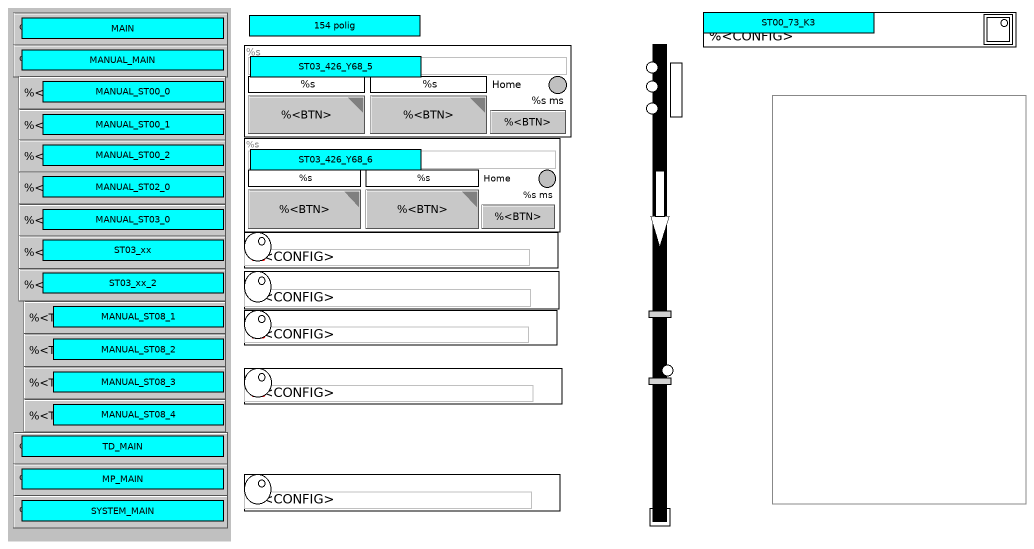
[picture p118: MANUAL_ST03_4 (HMI screen)]
embedded screen at (3,115)-(226,648): M0000_Manual
embedded screen at (239,152)-(566,244): ZLIB_VALVE_1_SENSORS
embedded screen at (239,245)-(555,339): ZLIB_VALVE_1_SENSORS
embedded screen at (239,417)-(552,452): VDIGIN
embedded screen at (239,339)-(553,375): VDIGIN
embedded screen at (239,378)-(554,416): VDIGIN
embedded screen at (239,581)-(555,618): VDIGIN
embedded screen at (239,475)-(557,511): VDIGIN
embedded screen at (636,151)-(677,633): ZUFUEHRUNG_154POL; invisible if gTypeCode<>4871
rectangle at (244,122)-(415,143): text "154 polig"; invisible if TRUE
rectangle at (245,163)-(416,184): text "ST03_426_Y68_5"; invisible if TRUE
rectangle at (245,256)-(416,277): text "ST03_426_Y68_6"; invisible if TRUE
embedded screen at (698,119)-(1011,154): VDIGOUT_SMAL
rectangle at (698,119)-(869,140): text "ST00_73_K3"; invisible if TRUE
1 more shapes without text or variables
*)

(* Visualisation MANUAL_ST03_5
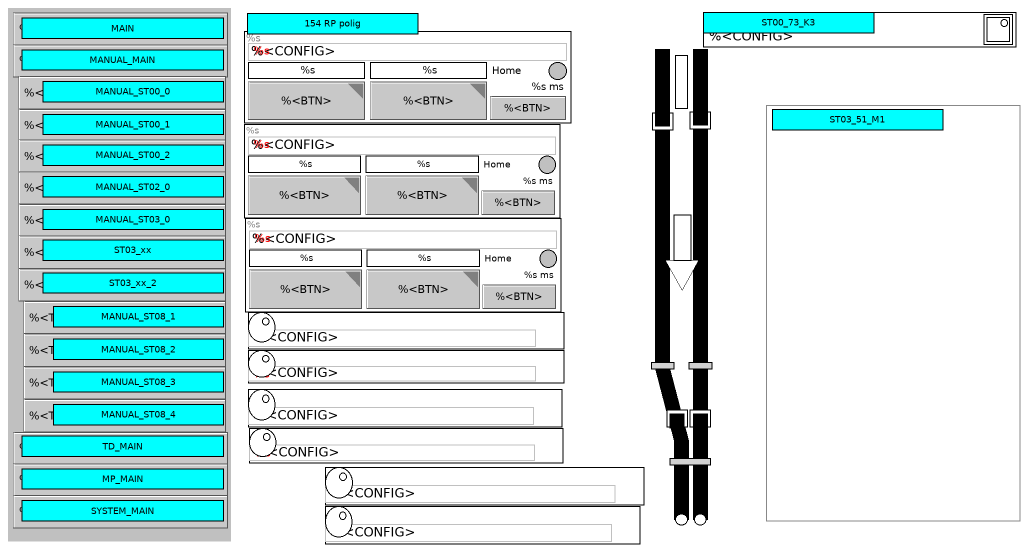
embedded screen at (3,115)-(226,648): M0000_Manual
embedded screen at (239,138)-(566,230): ZLIB_VALVE_1_SENSORS
embedded screen at (239,231)-(555,325): ZLIB_VALVE_1_SENSORS
embedded screen at (244,535)-(558,570): VDIGIN
embedded screen at (320,574)-(639,612): VDIGIN
embedded screen at (243,457)-(559,490): VDIGIN
embedded screen at (243,496)-(557,534): VDIGIN
embedded screen at (243,419)-(559,456): VDIGIN
embedded screen at (320,613)-(635,651): VDIGIN
embedded screen at (240,325)-(556,419): ZLIB_VALVE_1_SENSORS
embedded screen at (646,156)-(707,632): ZUFUEHRUNG_154RP; invisible if gTypeCode<>4872
rectangle at (242,120)-(413,141): text "154 RP polig"; invisible if TRUE
rectangle at (767,216)-(938,237): text "ST03_51_M1"; invisible if TRUE
embedded screen at (698,119)-(1011,154): VDIGOUT_SMAL
rectangle at (698,119)-(869,140): text "ST00_73_K3"; invisible if TRUE
1 more shapes without text or variables
*)

(* Visualisation MANUAL_ST03_6
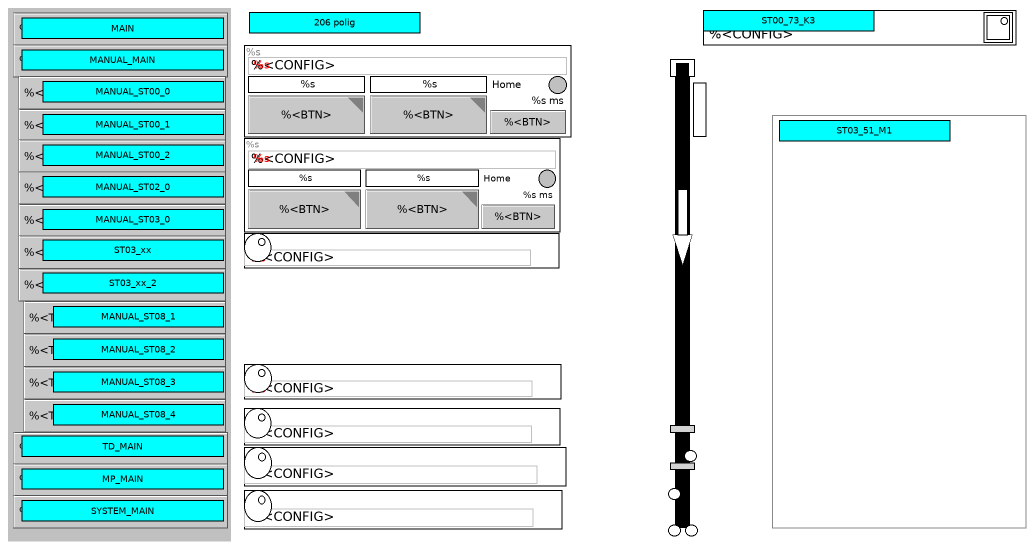
embedded screen at (3,115)-(226,648): M0000_Manual
embedded screen at (239,152)-(566,244): ZLIB_VALVE_1_SENSORS
embedded screen at (239,245)-(555,339): ZLIB_VALVE_1_SENSORS
embedded screen at (239,554)-(561,593): VDIGIN
embedded screen at (239,340)-(554,375): VDIGIN
embedded screen at (239,515)-(555,552): VDIGIN
embedded screen at (239,597)-(557,636): VDIGIN
embedded screen at (239,471)-(556,506): VDIGIN
embedded screen at (646,161)-(701,643): ZUFUEHRUNG_206POL; invisible if gTypeCode<>522
rectangle at (244,119)-(415,140): text "206 polig"; invisible if TRUE
rectangle at (774,227)-(945,248): text "ST03_51_M1"; invisible if TRUE
embedded screen at (698,117)-(1011,152): VDIGOUT_SMAL
rectangle at (698,117)-(869,138): text "ST00_73_K3"; invisible if TRUE
1 more shapes without text or variables
*)

(* Visualisation MANUAL_ST03_7
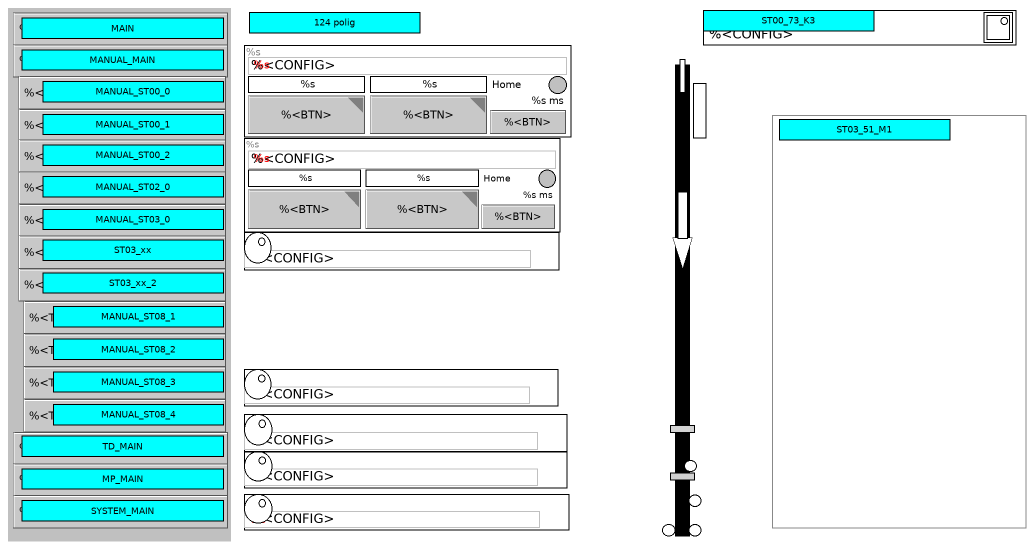
embedded screen at (3,115)-(226,648): M0000_Manual
embedded screen at (239,152)-(566,244): ZLIB_VALVE_1_SENSORS
embedded screen at (239,245)-(555,339): ZLIB_VALVE_1_SENSORS
embedded screen at (239,558)-(562,595): VDIGIN
embedded screen at (239,339)-(554,377): VDIGIN
embedded screen at (239,521)-(562,559): VDIGIN
embedded screen at (239,601)-(564,637): VDIGIN
embedded screen at (239,476)-(553,513): VDIGIN
embedded screen at (646,161)-(701,643): ZUFUEHRUNG_124POL; invisible if gTypeCode<>564
rectangle at (244,119)-(415,140): text "124 polig"; invisible if TRUE
rectangle at (774,226)-(945,247): text "ST03_51_M1"; invisible if TRUE
embedded screen at (698,117)-(1011,152): VDIGOUT_SMAL
rectangle at (698,117)-(869,138): text "ST00_73_K3"; invisible if TRUE
1 more shapes without text or variables
*)

(* Visualisation MANUAL_ST03_8
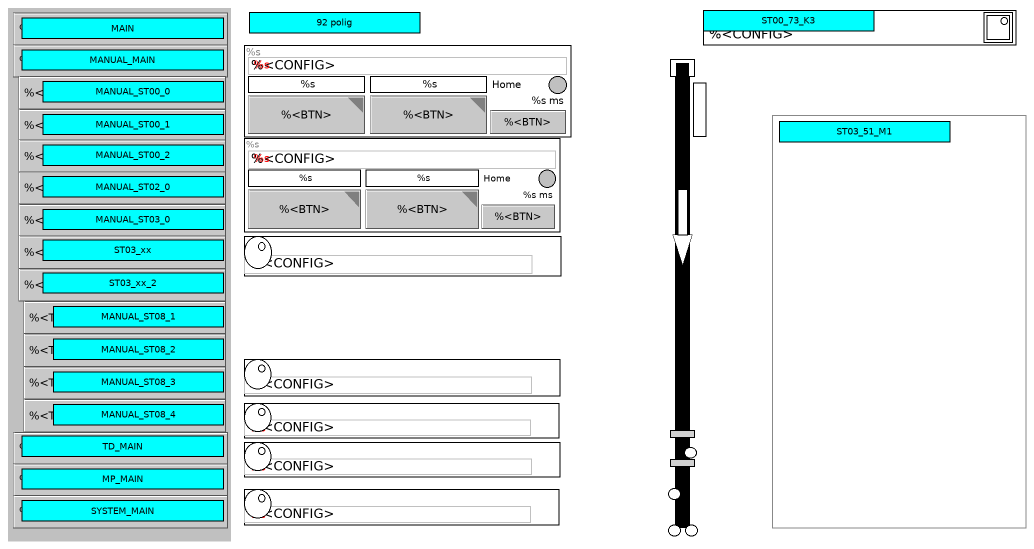
embedded screen at (3,115)-(226,648): M0000_Manual
embedded screen at (239,152)-(566,244): ZLIB_VALVE_1_SENSORS
embedded screen at (239,245)-(555,339): ZLIB_VALVE_1_SENSORS
embedded screen at (239,549)-(555,584): VDIGIN
embedded screen at (239,343)-(556,383): VDIGIN
embedded screen at (239,510)-(554,545): VDIGIN
embedded screen at (239,596)-(554,632): VDIGIN
embedded screen at (239,466)-(555,503): VDIGIN
embedded screen at (646,161)-(701,643): ZUFUEHRUNG_92POL; invisible if gTypeCode<>550
rectangle at (244,119)-(415,140): text "92 polig"; invisible if TRUE
rectangle at (774,228)-(945,249): text "ST03_51_M1"; invisible if TRUE
embedded screen at (698,117)-(1011,152): VDIGOUT_SMAL
rectangle at (698,117)-(869,138): text "ST00_73_K3"; invisible if TRUE
1 more shapes without text or variables
*)

(* Visualisation MANUAL_ST03_9
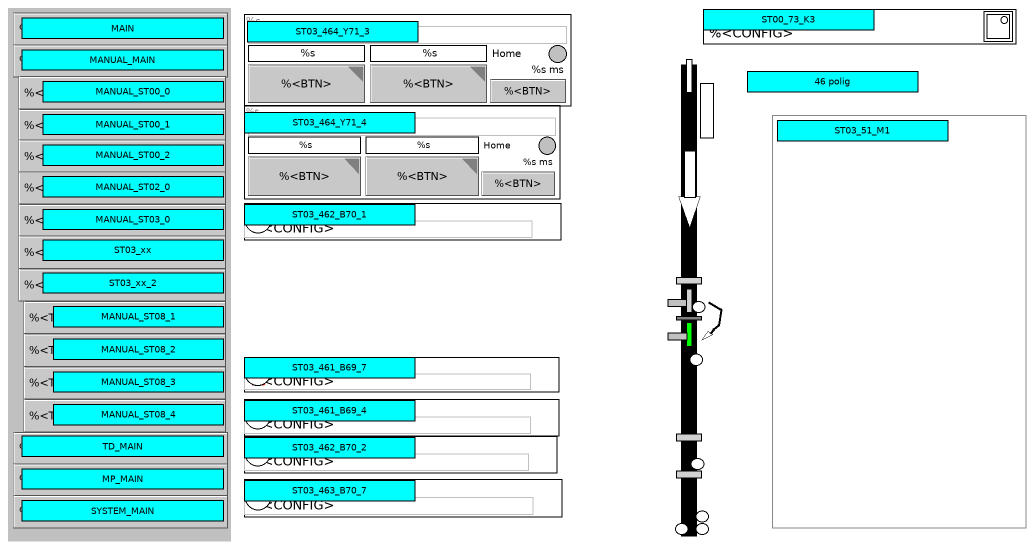
embedded screen at (3,115)-(226,648): M0000_Manual
embedded screen at (239,121)-(566,213): ZLIB_VALVE_1_SENSORS
embedded screen at (239,212)-(555,306): ZLIB_VALVE_1_SENSORS
embedded screen at (239,543)-(552,580): VDIGIN
embedded screen at (239,310)-(556,347): VDIGIN
embedded screen at (239,506)-(554,543): VDIGIN
embedded screen at (239,586)-(557,624): VDIGIN
embedded screen at (239,464)-(554,499): VDIGIN
embedded screen at (646,161)-(716,643): ZUFUEHRUNG_46POL; invisible if gTypeCode<>569
rectangle at (742,178)-(913,199): text "46 polig"; invisible if TRUE
rectangle at (239,219)-(410,240): text "ST03_464_Y71_4"; invisible if TRUE
rectangle at (242,128)-(413,149): text "ST03_464_Y71_3"; invisible if TRUE
rectangle at (239,311)-(410,332): text "ST03_462_B70_1"; invisible if TRUE
rectangle at (239,507)-(410,528): text "ST03_461_B69_4"; invisible if TRUE
rectangle at (239,544)-(410,565): text "ST03_462_B70_2"; invisible if TRUE
rectangle at (239,587)-(410,608): text "ST03_463_B70_7"; invisible if TRUE
rectangle at (239,464)-(410,485): text "ST03_461_B69_7"; invisible if TRUE
rectangle at (772,227)-(943,248): text "ST03_51_M1"; invisible if TRUE
embedded screen at (698,116)-(1011,151): VDIGOUT_SMAL
rectangle at (698,116)-(869,137): text "ST00_73_K3"; invisible if TRUE
1 more shapes without text or variables
*)

(* Visualisation MANUAL_ST03_9_2
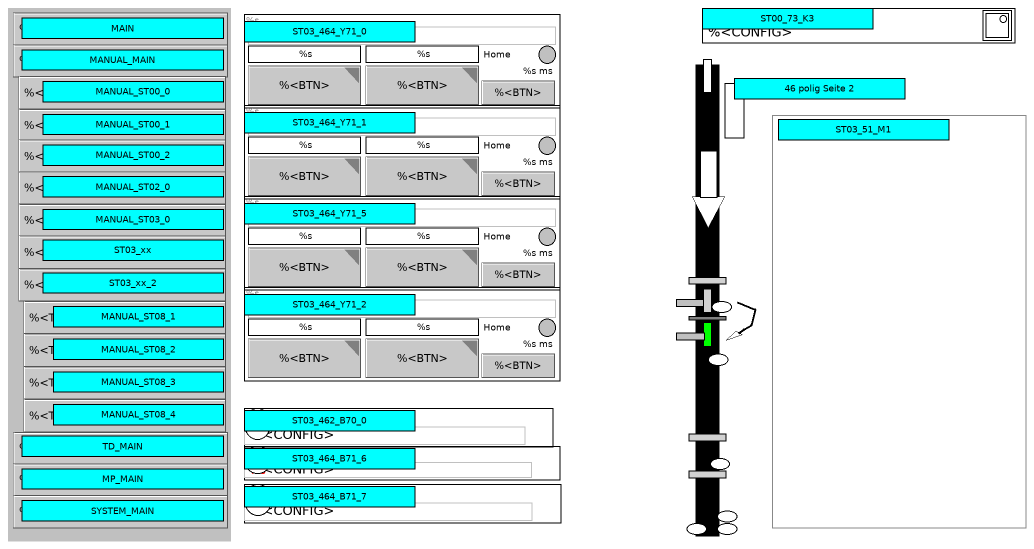
embedded screen at (3,115)-(226,648): M0000_Manual
embedded screen at (646,161)-(750,643): ZUFUEHRUNG_46POL; invisible if gTypeCode<>569
rectangle at (729,185)-(900,206): text "46 polig Seite 2"; invisible if TRUE
embedded screen at (239,553)-(555,587): VDIGIN
embedded screen at (239,121)-(555,215): ZLIB_VALVE_1_SENSORS
rectangle at (239,128)-(410,149): text "ST03_464_Y71_0"; invisible if TRUE
rectangle at (239,555)-(410,576): text "ST03_464_B71_6"; invisible if TRUE
embedded screen at (239,212)-(555,306): ZLIB_VALVE_1_SENSORS
rectangle at (239,219)-(410,240): text "ST03_464_Y71_1"; invisible if TRUE
embedded screen at (239,394)-(555,488): ZLIB_VALVE_1_SENSORS
rectangle at (239,401)-(410,422): text "ST03_464_Y71_2"; invisible if TRUE
embedded screen at (239,303)-(555,397): ZLIB_VALVE_1_SENSORS
rectangle at (239,310)-(410,331): text "ST03_464_Y71_5"; invisible if TRUE
embedded screen at (239,515)-(548,554): VDIGIN
rectangle at (239,517)-(410,538): text "ST03_462_B70_0"; invisible if TRUE
rectangle at (773,226)-(944,247): text "ST03_51_M1"; invisible if TRUE
embedded screen at (239,591)-(556,630): VDIGIN
rectangle at (239,593)-(410,614): text "ST03_464_B71_7"; invisible if TRUE
embedded screen at (697,115)-(1010,150): VDIGOUT_SMAL
rectangle at (697,115)-(868,136): text "ST00_73_K3"; invisible if TRUE
1 more shapes without text or variables
*)

(* Visualisation MANUAL_ST08_1
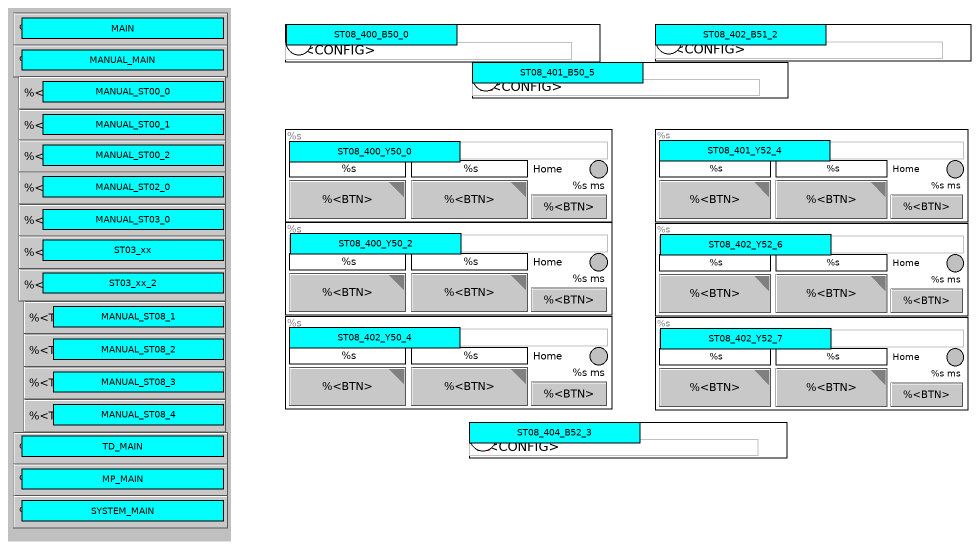
embedded screen at (3,115)-(226,648): M0000_Manual
embedded screen at (280,236)-(607,329): ZLIB_VALVE_1_SENSORS; invisible if NOT .MP.ST08.Trayzufuhr_Verlaengerung
embedded screen at (280,329)-(607,422): ZLIB_VALVE_1_SENSORS
embedded screen at (280,131)-(595,169): VDIGIN
embedded screen at (467,169)-(783,205): VDIGIN
embedded screen at (650,131)-(966,168): VDIGIN
embedded screen at (280,423)-(607,516): ZLIB_VALVE_1_SENSORS
embedded screen at (650,236)-(963,329): ZLIB_VALVE_1_SENSORS; invisible if NOT .MP.ST08.Traystapel_schieben OR NOT .MP.ST08.Trayzufuhr_Verlaengerung
embedded screen at (650,330)-(963,423): ZLIB_VALVE_1_SENSORS; invisible if NOT .MP.ST08.Traystapel_schieben OR NOT .MP.ST08.Trayzufuhr_Verlaengerung
embedded screen at (650,424)-(963,517): ZLIB_VALVE_1_SENSORS; invisible if NOT .MP.ST08.Traystapel_schieben
embedded screen at (464,529)-(782,565): VDIGIN
rectangle at (281,131)-(452,152): text "ST08_400_B50_0"; invisible if TRUE
rectangle at (467,169)-(638,190): text "ST08_401_B50_5"; invisible if TRUE
rectangle at (650,131)-(821,152): text "ST08_402_B51_2"; invisible if TRUE
rectangle at (284,248)-(455,269): text "ST08_400_Y50_0"; invisible if TRUE
rectangle at (285,340)-(456,361): text "ST08_400_Y50_2"; invisible if TRUE
rectangle at (654,247)-(825,268): text "ST08_401_Y52_4"; invisible if TRUE
rectangle at (655,341)-(826,362): text "ST08_402_Y52_6"; invisible if TRUE
rectangle at (655,435)-(826,456): text "ST08_402_Y52_7"; invisible if TRUE
rectangle at (284,434)-(455,455): text "ST08_402_Y50_4"; invisible if TRUE
rectangle at (464,529)-(635,550): text "ST08_404_B52_3"; invisible if TRUE
*)

(* Visualisation MANUAL_ST08_2
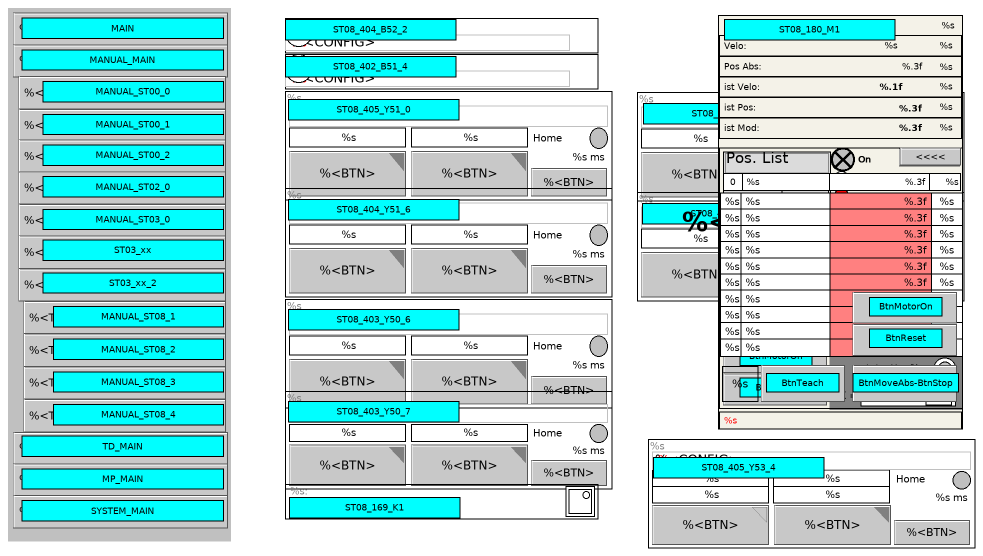
embedded screen at (3,115)-(226,648): M0000_Manual
embedded screen at (280,125)-(593,160): VDIGIN
embedded screen at (280,198)-(607,307): ZLIB_VALVE_1_SENSORS
embedded screen at (280,295)-(607,404): ZLIB_VALVE_1_SENSORS
embedded screen at (643,546)-(970,655): ZLIB_VALVE_2_SENSORS
embedded screen at (280,406)-(607,515): ZLIB_VALVE_1_SENSORS
embedded screen at (280,498)-(607,596): ZLIB_VALVE_1_SENSORS
embedded screen at (280,161)-(593,196): VDIGIN
embedded screen at (632,199)-(959,308): ZLIB_VALVE_1_SENSORS; invisible if MP.ST08.StapelMotor
rectangle at (638,210)-(809,231): text "ST08_404_Y53_0"; invisible if TRUE
embedded screen at (632,299)-(959,408): ZLIB_VALVE_1_SENSORS; invisible if MP.ST08.StapelMotor
rectangle at (637,310)-(808,331): text "ST08_404_Y53_2"; invisible if TRUE
embedded screen at (713,122)-(959,536): ZLIB_7211_Achse; invisible if NOT MP.ST08.StapelMotor
embedded screen at (280,591)-(593,626): VDIGOUT_SMAL
rectangle at (280,126)-(451,147): text "ST08_404_B52_2"; invisible if TRUE
rectangle at (280,163)-(451,184): text "ST08_402_B51_4"; invisible if TRUE
rectangle at (283,206)-(454,227): text "ST08_405_Y51_0"; invisible if TRUE
rectangle at (283,306)-(454,327): text "ST08_404_Y51_6"; invisible if TRUE
rectangle at (283,416)-(454,437): text "ST08_403_Y50_6"; invisible if TRUE
rectangle at (283,508)-(454,529): text "ST08_403_Y50_7"; invisible if TRUE
rectangle at (284,604)-(455,625): text "ST08_169_K1"; invisible if TRUE
rectangle at (648,564)-(819,585): text "ST08_405_Y53_4"; invisible if TRUE
rectangle at (719,126)-(890,147): text "ST08_180_M1"; invisible if TRUE
*)

(* Visualisation MANUAL_ST08_3
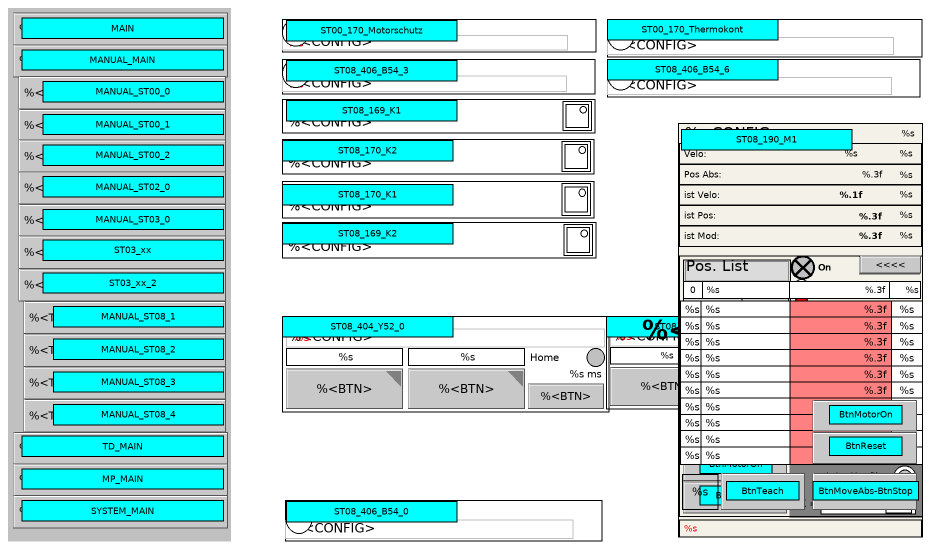
embedded screen at (3,115)-(226,648): M0000_Manual
embedded screen at (277,206)-(590,240): VDIGOUT_SMAL
embedded screen at (277,329)-(591,365): VDIGOUT_SMAL
embedded screen at (277,288)-(589,325): VDIGOUT_SMAL
embedded screen at (277,246)-(589,281): VDIGOUT_SMAL
embedded screen at (602,126)-(917,164): VDIGIN
embedded screen at (277,126)-(591,159): VDIGIN
embedded screen at (280,607)-(597,648): VDIGIN
embedded screen at (277,166)-(590,201): VDIGIN
embedded screen at (601,423)-(914,516): ZLIB_VALVE_1_SENSORS; invisible if MP.ST08.TrayAushebenMotor
embedded screen at (277,423)-(604,519): ZLIB_VALVE_1_SENSORS
rectangle at (601,423)-(772,444): text "ST08_406_Y52_3"; invisible if TRUE
rectangle at (277,423)-(448,444): text "ST08_404_Y52_0"; invisible if TRUE
rectangle at (281,207)-(452,228): text "ST08_169_K1"; invisible if TRUE
rectangle at (277,330)-(448,351): text "ST08_169_K2"; invisible if TRUE
rectangle at (277,291)-(448,312): text "ST08_170_K1"; invisible if TRUE
rectangle at (277,247)-(448,268): text "ST08_170_K2"; invisible if TRUE
rectangle at (281,127)-(452,148): text "ST00_170_Motorschutz"; invisible if TRUE
rectangle at (602,126)-(773,147): text "ST00_170_Thermokont"; invisible if TRUE
rectangle at (281,608)-(452,629): text "ST08_406_B54_0"; invisible if TRUE
rectangle at (281,167)-(452,188): text "ST08_406_B54_3"; invisible if TRUE
embedded screen at (602,166)-(915,204): VDIGIN
rectangle at (602,166)-(773,187): text "ST08_406_B54_6"; invisible if TRUE
embedded screen at (673,230)-(919,644): ZLIB_7211_Achse; invisible if NOT MP.ST08.TrayAushebenMotor
rectangle at (676,236)-(847,257): text "ST08_190_M1"; invisible if TRUE
*)

(* Visualisation MANUAL_ST08_4
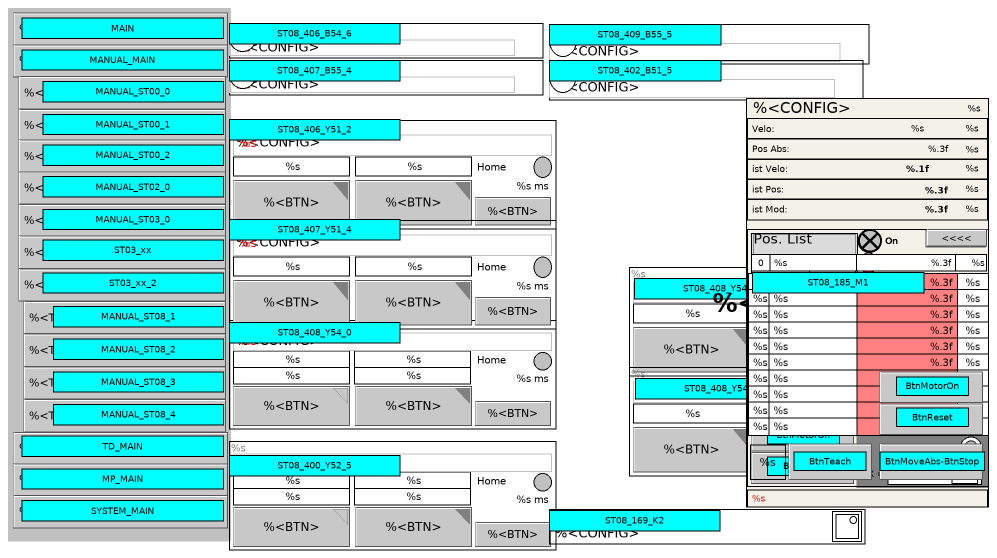
embedded screen at (3,115)-(226,648): M0000_Manual
embedded screen at (224,427)-(551,536): ZLIB_VALVE_2_SENSORS
embedded screen at (224,130)-(538,165): VDIGIN
embedded screen at (224,227)-(551,336): ZLIB_VALVE_1_SENSORS
embedded screen at (224,327)-(551,436): ZLIB_VALVE_1_SENSORS
embedded screen at (544,131)-(864,171): VDIGIN
embedded screen at (224,548)-(551,657): ZLIB_VALVE_2_SENSORS; invisible if MP.ST03.SGM_3621
embedded screen at (544,167)-(858,207): VDIGIN
embedded screen at (624,374)-(951,483): ZLIB_VALVE_1_SENSORS; invisible if MP.ST08.StapelMotor
rectangle at (629,385)-(801,406): text "ST08_408_Y54_2"; invisible if TRUE
embedded screen at (624,474)-(951,583): ZLIB_VALVE_1_SENSORS; invisible if MP.ST08.StapelMotor
rectangle at (630,485)-(802,506): text "ST08_408_Y54_4"; invisible if TRUE
embedded screen at (741,205)-(985,614): ZLIB_7211_Achse; invisible if NOT MP.ST08.StapelMotor
embedded screen at (224,167)-(538,202): VDIGIN
embedded screen at (544,616)-(860,651): VDIGOUT_SMAL
rectangle at (224,562)-(395,583): text "ST08_400_Y52_5"; invisible if TRUE
rectangle at (544,617)-(715,638): text "ST08_169_K2"; invisible if TRUE
rectangle at (224,429)-(395,450): text "ST08_408_Y54_0"; invisible if TRUE
rectangle at (224,326)-(395,347): text "ST08_407_Y51_4"; invisible if TRUE
rectangle at (224,226)-(395,247): text "ST08_406_Y51_2"; invisible if TRUE
rectangle at (224,130)-(395,151): text "ST08_406_B54_6"; invisible if TRUE
rectangle at (224,167)-(395,188): text "ST08_407_B55_4"; invisible if TRUE
rectangle at (544,131)-(716,152): text "ST08_409_B55_5"; invisible if TRUE
rectangle at (544,167)-(716,188): text "ST08_402_B51_5"; invisible if TRUE
rectangle at (747,379)-(919,400): text "ST08_185_M1"; invisible if TRUE
*)

(* Visualisation DIALOG_SAVE_AS
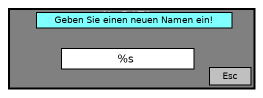
rectangle at (1,0)-(248,81): text "%<DATA>"; shows 'save_as'
rectangle at (54,40)-(187,61): text "%s"; shows $InputVar$; invisible if ( *NOT ST_TD.b_Dialog_save_as_on* ); editable
rectangle at (29,4)-(225,20): text "Geben Sie einen neuen Namen ein!"; invisible if TRUE
rectangle at (202,59)-(244,77): text "Esc"; toggles TDHandler.b_Dialog_save_as_on
*)

(* Visualisation TD_01_EDIT
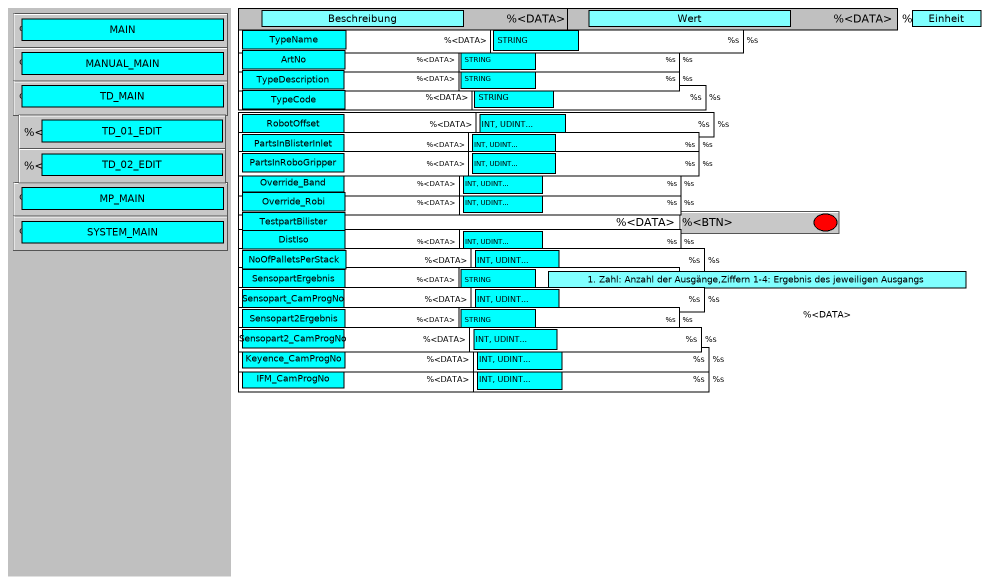
embedded screen at (3,115)-(226,683): M0003_TD
rectangle at (796,407)-(1009,436): text "%<DATA>"; shows 'Info_01'; invisible if gTypeCode<>4991 AND gTypeCode <>312
embedded screen at (233,317)-(834,342): Data_BOOL
embedded screen at (233,192)-(870,217): Data_STRING
embedded screen at (233,297)-(834,322): Data_DEZIMAL
embedded screen at (233,278)-(834,303): Data_DEZIMAL
embedded screen at (233,173)-(834,198): Data_STRING
embedded screen at (233,154)-(834,179): Data_STRING
embedded screen at (233,135)-(921,160): Data_STRING
embedded screen at (233,336)-(834,361): Data_DEZIMAL
embedded screen at (233,355)-(866,380): Data_DEZIMAL
embedded screen at (233,374)-(834,399): Data_STRING
rectangle at (237,137)-(341,156): text "TypeName"; invisible if TRUE
rectangle at (237,157)-(340,176): text "ArtNo"; invisible if TRUE
rectangle at (237,177)-(339,196): text "TypeDescription"; invisible if TRUE
rectangle at (237,197)-(340,216): text "TypeCode"; invisible if TRUE
rectangle at (237,280)-(339,299): text "Override_Band"; invisible if TRUE
rectangle at (237,299)-(340,318): text "Override_Robi"; invisible if TRUE
rectangle at (237,319)-(340,338): text "TestpartBilister"; invisible if TRUE
rectangle at (237,337)-(340,356): text "DistIso"; invisible if TRUE
rectangle at (237,376)-(340,395): text "SensopartErgebnis"; invisible if TRUE
rectangle at (237,357)-(341,376): text "NoOfPalletsPerStack"; invisible if TRUE
rectangle at (543,378)-(961,395): text "1. Zahl: Anzahl der Ausgänge,Ziffern 1-4: Ergebnis des jeweiligen Ausgangs"; invisible if TRUE
embedded screen at (233,219)-(879,244): Data_DEZIMAL
rectangle at (237,221)-(339,240): text "RobotOffset"; invisible if TRUE
embedded screen at (233,239)-(859,264): Data_DEZIMAL
rectangle at (237,241)-(339,260): text "PartsInBlisterInlet"; invisible if TRUE
embedded screen at (233,474)-(872,499): Data_DEZIMAL
rectangle at (237,476)-(339,495): text "IFM_CamProgNo"; invisible if TRUE
embedded screen at (233,394)-(866,419): Data_DEZIMAL
rectangle at (237,396)-(339,415): text "Sensopart_CamProgNo"; invisible if TRUE
embedded screen at (233,258)-(859,283): Data_DEZIMAL
rectangle at (237,260)-(339,279): text "PartsInRoboGripper"; invisible if TRUE
embedded screen at (233,115)-(987,137): DATA_HEADER_BEER
embedded screen at (233,454)-(872,479): Data_DEZIMAL
rectangle at (237,456)-(340,475): text "Keyence_CamProgNo"; invisible if TRUE
embedded screen at (233,414)-(834,439): Data_STRING
rectangle at (237,416)-(340,435): text "Sensopart2Ergebnis"; invisible if TRUE
embedded screen at (233,434)-(862,459): Data_DEZIMAL
rectangle at (237,436)-(339,455): text "Sensopart2_CamProgNo"; invisible if TRUE
*)

(* Visualisation TD_02_EDIT
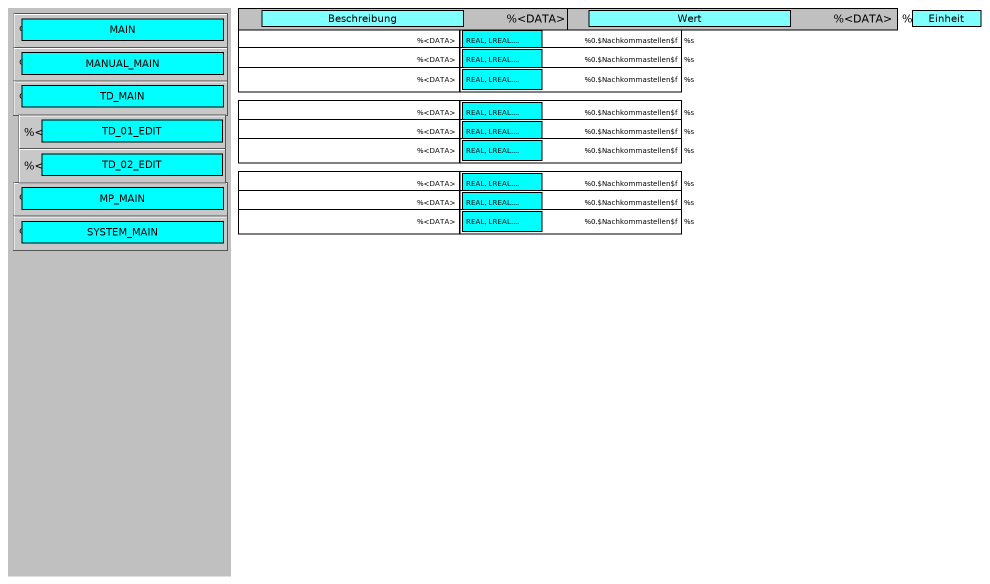
embedded screen at (3,115)-(226,683): M0003_TD
embedded screen at (233,135)-(834,160): Data_DEZIMAL_REAL
embedded screen at (233,154)-(834,179): Data_DEZIMAL_REAL
embedded screen at (233,174)-(834,199): Data_DEZIMAL_REAL
embedded screen at (233,207)-(834,232): Data_DEZIMAL_REAL
embedded screen at (233,226)-(834,251): Data_DEZIMAL_REAL
embedded screen at (233,245)-(834,270): Data_DEZIMAL_REAL
embedded screen at (233,115)-(987,137): DATA_HEADER_BEER
embedded screen at (233,278)-(834,303): Data_DEZIMAL_REAL
embedded screen at (233,297)-(834,322): Data_DEZIMAL_REAL
embedded screen at (233,316)-(834,341): Data_DEZIMAL_REAL
*)

(* Visualisation TD_MAIN
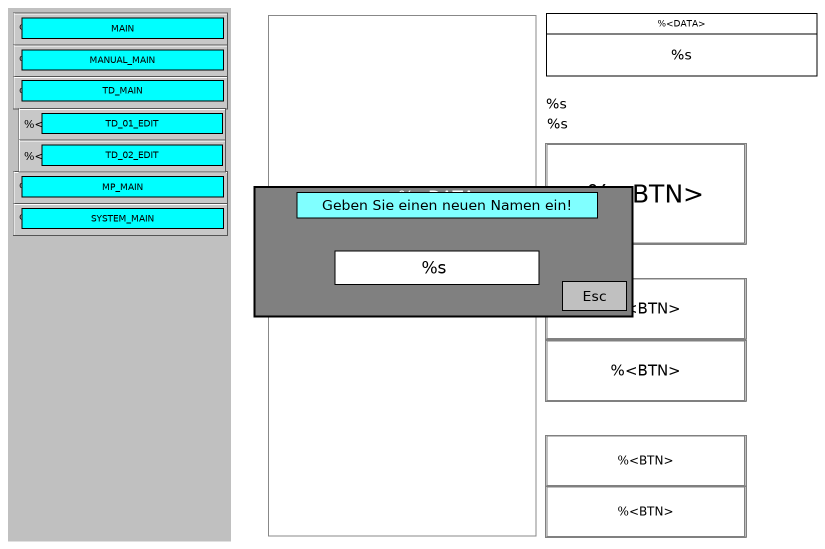
rectangle at (541,140)-(812,183): text "%s"; shows .sTDHandler.FileFilter; editable
rectangle at (541,120)-(812,141): text "%<DATA>"; shows 'Filter'
embedded screen at (540,250)-(741,351): ZLIB_VISUBUTTON
embedded screen at (540,447)-(741,508): ZLIB_VISUBUTTON
embedded screen at (3,115)-(226,648): M0003_TD
embedded screen at (540,542)-(741,593): ZLIB_VISUBUTTON
embedded screen at (540,593)-(741,644): ZLIB_VISUBUTTON
embedded screen at (540,385)-(741,446): ZLIB_VISUBUTTON
embedded screen at (247,293)-(628,424): DIALOG_SAVE_AS; invisible if NOT TDHandler.b_Dialog_save_as_on
rectangle at (539,200)-(730,221): text "%s"; shows TDHandler.s_Typecode
rectangle at (540,220)-(731,241): text "%s"; shows TDHandler.s_Typedescription
1 more shapes without text or variables
*)

(* Visualisation MP_DATE
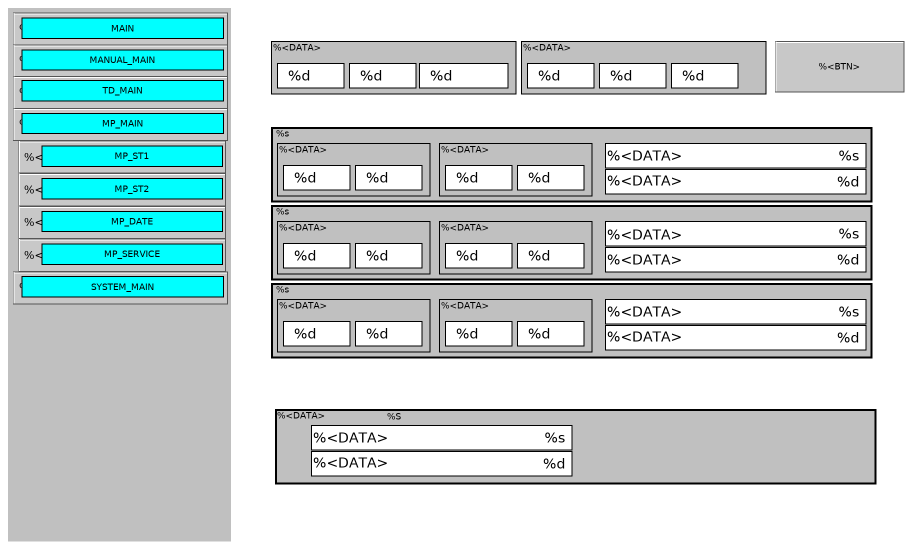
rectangle at (266,390)-(867,465): text "%s"; shows .MP.ShiftData.Shift[3].ShiftName; alarm colour if .MP.ShiftData.Shift[3].ShiftActive
rectangle at (266,312)-(867,387): text "%s"; shows .MP.ShiftData.Shift[2].ShiftName; alarm colour if .MP.ShiftData.Shift[2].ShiftActive
rectangle at (266,234)-(867,309): text "%s"; shows .MP.ShiftData.Shift[1].ShiftName; alarm colour if .MP.ShiftData.Shift[1].ShiftActive
rectangle at (516,148)-(761,201): text "%<DATA>"; shows 'Uhrzeit'
rectangle at (266,148)-(511,201): text "%<DATA>"; shows 'Datum'
embedded screen at (3,115)-(226,648): M0002_Machpara
rectangle at (272,170)-(339,195): text "%d"; shows CallGeneralFunctions.SetTimeStruct.wDay; editable 1..31
rectangle at (344,170)-(411,195): text "%d"; shows CallGeneralFunctions.SetTimeStruct.wMonth; editable 1..12
rectangle at (414,170)-(503,195): text "%d"; shows CallGeneralFunctions.SetTimeStruct.wYear; editable 2000..3000
rectangle at (522,170)-(589,195): text "%d"; shows CallGeneralFunctions.SetTimeStruct.wHour; editable 0..24
rectangle at (594,170)-(661,195): text "%d"; shows CallGeneralFunctions.SetTimeStruct.wMinute; editable 0..59
rectangle at (666,170)-(733,195): text "%d"; shows CallGeneralFunctions.SetTimeStruct.wSecond; editable 0..59
button at (770,148)-(899,199): text "%<BTN>"; shows 'set Clock'; taps CallGeneralFunctions.SetLocalTime.START; dynamic style Color.lightgrey
rectangle at (272,250)-(425,303): text "%<DATA>"; shows 'Uhrzeit Start'
rectangle at (278,272)-(345,297): text "%d"; shows .MP.ShiftData.Shift[1].TimeStart.wHour; editable 0..24
rectangle at (350,272)-(417,297): text "%d"; shows .MP.ShiftData.Shift[1].TimeStart.wMinute; editable 0..59
rectangle at (434,250)-(587,303): text "%<DATA>"; shows 'Uhrzeit Ende'
rectangle at (440,272)-(507,297): text "%d"; shows .MP.ShiftData.Shift[1].TimeEnd.wHour; editable 0..24
rectangle at (512,272)-(579,297): text "%d"; shows .MP.ShiftData.Shift[1].TimeEnd.wMinute; editable 0..59
rectangle at (272,328)-(425,381): text "%<DATA>"; shows 'Uhrzeit Start'
rectangle at (278,350)-(345,375): text "%d"; shows .MP.ShiftData.Shift[2].TimeStart.wHour; editable 0..24
rectangle at (350,350)-(417,375): text "%d"; shows .MP.ShiftData.Shift[2].TimeStart.wMinute; editable 0..59
rectangle at (434,328)-(587,381): text "%<DATA>"; shows 'Uhrzeit Ende'
rectangle at (440,350)-(507,375): text "%d"; shows .MP.ShiftData.Shift[2].TimeEnd.wHour; editable 0..24
rectangle at (512,350)-(579,375): text "%d"; shows .MP.ShiftData.Shift[2].TimeEnd.wMinute; editable 0..59
rectangle at (272,406)-(425,459): text "%<DATA>"; shows 'Uhrzeit Start'
rectangle at (278,428)-(345,453): text "%d"; shows .MP.ShiftData.Shift[3].TimeStart.wHour; editable 0..24
rectangle at (350,428)-(417,453): text "%d"; shows .MP.ShiftData.Shift[3].TimeStart.wMinute; editable 0..59
rectangle at (434,406)-(587,459): text "%<DATA>"; shows 'Uhrzeit Ende'
rectangle at (440,428)-(507,453): text "%d"; shows .MP.ShiftData.Shift[3].TimeEnd.wHour; editable 0..24
rectangle at (512,428)-(579,453): text "%d"; shows .MP.ShiftData.Shift[3].TimeEnd.wMinute; editable 0..59
rectangle at (270,516)-(871,591): text "%<DATA>"; shows 'Aktuelle Schicht'; alarm colour if .MP.ShiftData.Activeshift.ShiftActive
rectangle at (600,250)-(861,275): text "%s"; shows .MP.ShiftData.Shift[1].ShiftName; editable
rectangle at (600,276)-(861,301): text "%d"; shows .MP.ShiftData.Shift[1].ShiftIndex; editable 1..3
rectangle at (600,328)-(861,353): text "%s"; shows .MP.ShiftData.Shift[2].ShiftName; editable
rectangle at (600,354)-(861,379): text "%d"; shows .MP.ShiftData.Shift[2].ShiftIndex; editable 1..3
rectangle at (600,406)-(861,431): text "%s"; shows .MP.ShiftData.Shift[3].ShiftName; editable
rectangle at (600,432)-(861,457): text "%d"; shows .MP.ShiftData.Shift[3].ShiftIndex; editable 1..3
rectangle at (306,532)-(567,557): text "%s"; shows .MP.ShiftData.ActiveShift.ShiftName
rectangle at (306,558)-(567,583): text "%d"; shows .MP.ShiftData.ActiveShift.ShiftIndex
rectangle at (380,515)-(511,532): text "%S"; shows .MP.ShiftData.Activeshift.ShiftName
rectangle at (306,532)-(521,557): text "%<DATA>"; shows 'Schicht Name'
rectangle at (306,557)-(522,582): text "%<DATA>"; shows 'Schicht Nummer'
rectangle at (600,406)-(815,431): text "%<DATA>"; shows 'Schicht Name'
rectangle at (600,431)-(816,456): text "%<DATA>"; shows 'Schicht Nummer'
rectangle at (600,329)-(815,354): text "%<DATA>"; shows 'Schicht Name'
rectangle at (600,354)-(816,379): text "%<DATA>"; shows 'Schicht Nummer'
rectangle at (600,250)-(815,275): text "%<DATA>"; shows 'Schicht Name'
rectangle at (600,275)-(816,300): text "%<DATA>"; shows 'Schicht Nummer'
*)

(* Visualisation MP_SERVICE
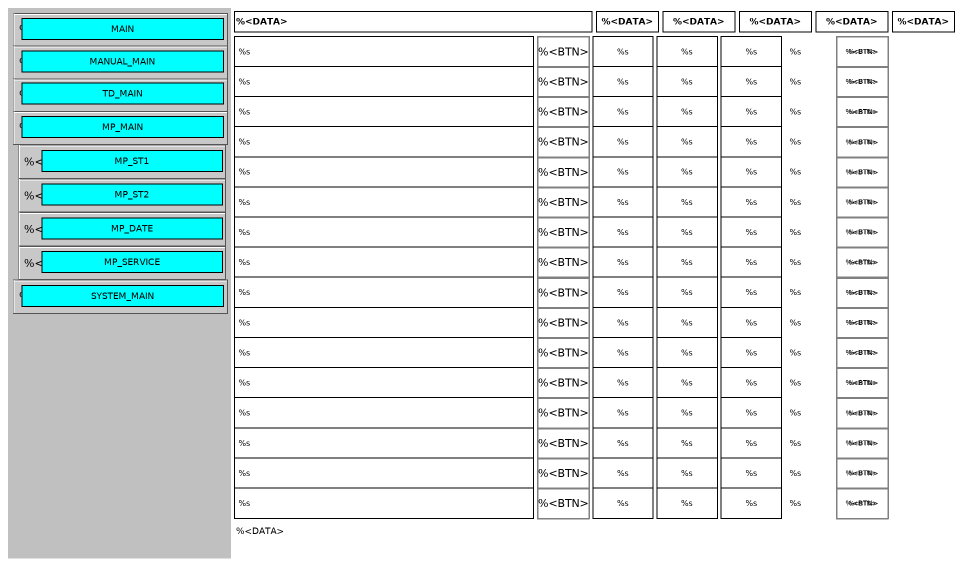
embedded screen at (3,115)-(226,665): M0002_Machpara
embedded screen at (229,118)-(1011,651): ZLIB_SERVICELIST
*)

(* Visualisation MP_ST1
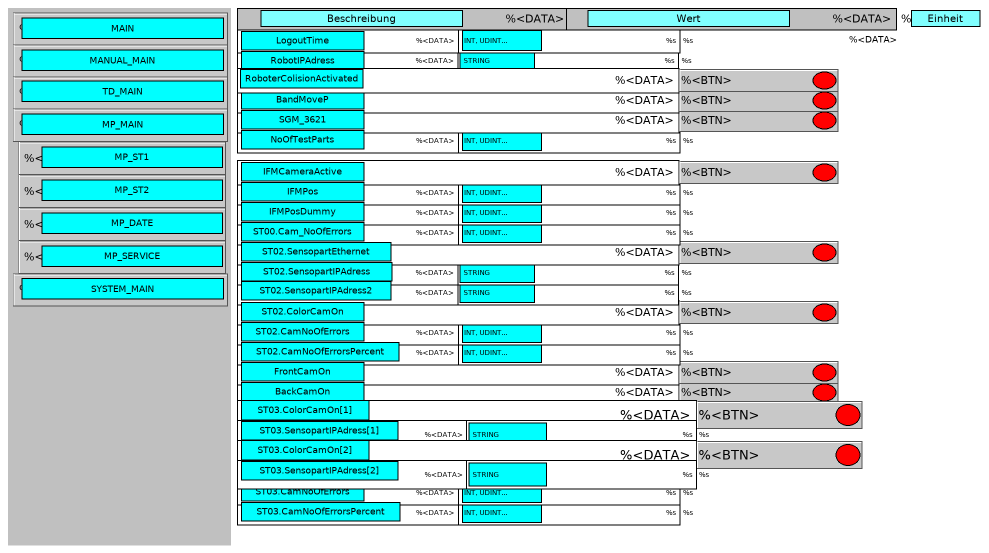
embedded screen at (3,115)-(226,652): M0002_Machpara
rectangle at (842,136)-(960,157): text "%<DATA>"; shows '0_deaktiv'
embedded screen at (232,607)-(833,632): Data_DEZIMAL
embedded screen at (232,587)-(833,612): Data_DEZIMAL
embedded screen at (232,487)-(833,512): Data_BOOL; dynamic style ST_CPU.LNG <> 2
embedded screen at (232,467)-(833,492): Data_BOOL; dynamic style ST_CPU.LNG <> 2
embedded screen at (232,447)-(833,472): Data_DEZIMAL
embedded screen at (232,427)-(833,452): Data_DEZIMAL
embedded screen at (232,407)-(833,432): Data_BOOL; dynamic style ST_CPU.LNG <> 2
embedded screen at (232,387)-(833,412): Data_STRING
embedded screen at (232,367)-(833,392): Data_STRING
embedded screen at (232,347)-(833,372): Data_BOOL
embedded screen at (232,327)-(833,352): Data_DEZIMAL
embedded screen at (232,307)-(833,332): Data_DEZIMAL
embedded screen at (232,287)-(833,312): Data_DEZIMAL
embedded screen at (232,267)-(833,292): Data_BOOL; dynamic style TRUE
embedded screen at (232,235)-(833,260): Data_DEZIMAL
embedded screen at (232,215)-(833,240): Data_BOOL
embedded screen at (232,195)-(833,220): Data_BOOL
embedded screen at (232,155)-(833,180): Data_STRING
embedded screen at (232,135)-(833,160): Data_DEZIMAL
rectangle at (236,158)-(359,177): text "RobotIPAdress"; invisible if TRUE
rectangle at (236,197)-(359,216): text "BandMoveP"; invisible if TRUE
rectangle at (236,217)-(359,236): text "SGM_3621"; invisible if TRUE
rectangle at (236,369)-(387,388): text "ST02.SensopartIPAdress"; invisible if TRUE
rectangle at (236,349)-(386,368): text "ST02.SensopartEthernet"; invisible if TRUE
rectangle at (236,269)-(359,288): text "IFMCameraActive"; invisible if TRUE
rectangle at (236,309)-(359,328): text "IFMPosDummy"; invisible if TRUE
rectangle at (236,388)-(386,407): text "ST02.SensopartIPAdress2"; invisible if TRUE
rectangle at (236,449)-(394,468): text "ST02.CamNoOfErrorsPercent"; invisible if TRUE
rectangle at (236,469)-(359,488): text "FrontCamOn"; invisible if TRUE
rectangle at (236,609)-(395,628): text "ST03.CamNoOfErrorsPercent"; invisible if TRUE
rectangle at (236,237)-(359,256): text "NoOfTestParts"; invisible if TRUE
rectangle at (236,329)-(359,348): text "ST00.Cam_NoOfErrors"; invisible if TRUE
rectangle at (236,429)-(359,448): text "ST02.CamNoOfErrors"; invisible if TRUE
rectangle at (236,489)-(359,508): text "BackCamOn"; shows 'BackCamOn'; invisible if TRUE
rectangle at (236,589)-(359,608): text "ST03.CamNoOfErrors"; invisible if TRUE
rectangle at (236,289)-(359,308): text "IFMPos"; invisible if TRUE
rectangle at (236,138)-(359,157): text "LogoutTime"; invisible if TRUE
rectangle at (236,409)-(359,428): text "ST02.ColorCamOn"; invisible if TRUE
embedded screen at (232,175)-(833,200): Data_BOOL
rectangle at (235,176)-(358,195): text "RoboterColisionActivated"; shows 'BackCamOn'; invisible if TRUE
embedded screen at (232,115)-(986,137): DATA_HEADER_BEER
embedded screen at (232,507)-(857,537): Data_BOOL
embedded screen at (232,527)-(857,556): Data_STRING
rectangle at (236,528)-(393,547): text "ST03.SensopartIPAdress[1]"; invisible if TRUE
rectangle at (236,507)-(364,527): text "ST03.ColorCamOn[1]"; invisible if TRUE
embedded screen at (232,547)-(857,577): Data_BOOL
embedded screen at (232,567)-(857,596): Data_STRING
rectangle at (236,568)-(393,587): text "ST03.SensopartIPAdress[2]"; invisible if TRUE
rectangle at (236,547)-(364,567): text "ST03.ColorCamOn[2]"; invisible if TRUE
*)

(* Visualisation MP_ST2
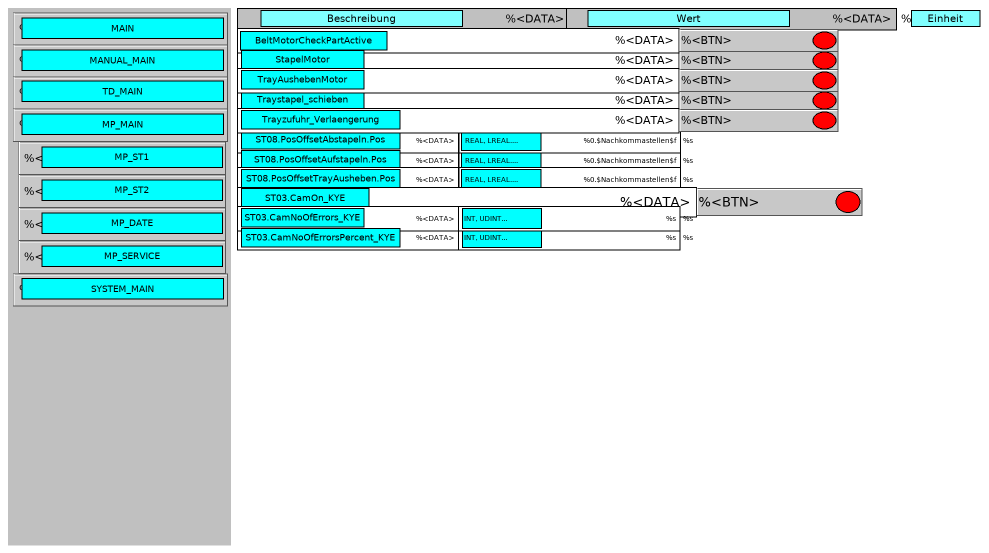
embedded screen at (3,115)-(226,652): M0002_Machpara
embedded screen at (232,115)-(986,137): DATA_HEADER_BEER
embedded screen at (232,255)-(833,280): Data_DEZIMAL_REAL
embedded screen at (232,235)-(833,260): Data_DEZIMAL_REAL
embedded screen at (232,195)-(833,220): Data_BOOL
embedded screen at (232,155)-(833,180): Data_BOOL
embedded screen at (232,135)-(833,160): Data_BOOL
rectangle at (236,197)-(359,216): text "Traystapel_schieben"; invisible if TRUE
rectangle at (236,157)-(359,176): text "StapelMotor"; invisible if TRUE
rectangle at (236,237)-(395,256): text "ST08.PosOffsetAbstapeln.Pos"; invisible if TRUE
rectangle at (236,257)-(395,276): text "ST08.PosOffsetAufstapeln.Pos"; invisible if TRUE
rectangle at (235,138)-(382,157): text "BeltMotorCheckPartActive"; invisible if TRUE
embedded screen at (232,175)-(833,200): Data_BOOL
rectangle at (236,177)-(359,196): text "TrayAushebenMotor"; invisible if TRUE
embedded screen at (232,274)-(833,299): Data_DEZIMAL_REAL
rectangle at (236,276)-(395,295): text "ST08.PosOffsetTrayAusheben.Pos"; invisible if TRUE
embedded screen at (232,215)-(833,240): Data_BOOL
rectangle at (236,217)-(395,236): text "Trayzufuhr_Verlaengerung"; invisible if TRUE
embedded screen at (232,294)-(857,324): Data_BOOL
rectangle at (236,295)-(364,315): text "ST03.CamOn_KYE"; invisible if TRUE
embedded screen at (232,332)-(833,357): Data_DEZIMAL
embedded screen at (232,313)-(833,338): Data_DEZIMAL
rectangle at (236,335)-(395,354): text "ST03.CamNoOfErrorsPercent_KYE"; invisible if TRUE
rectangle at (236,315)-(359,334): text "ST03.CamNoOfErrors_KYE"; invisible if TRUE
*)

(* Visualisation SYSTEM_ERRORLIST
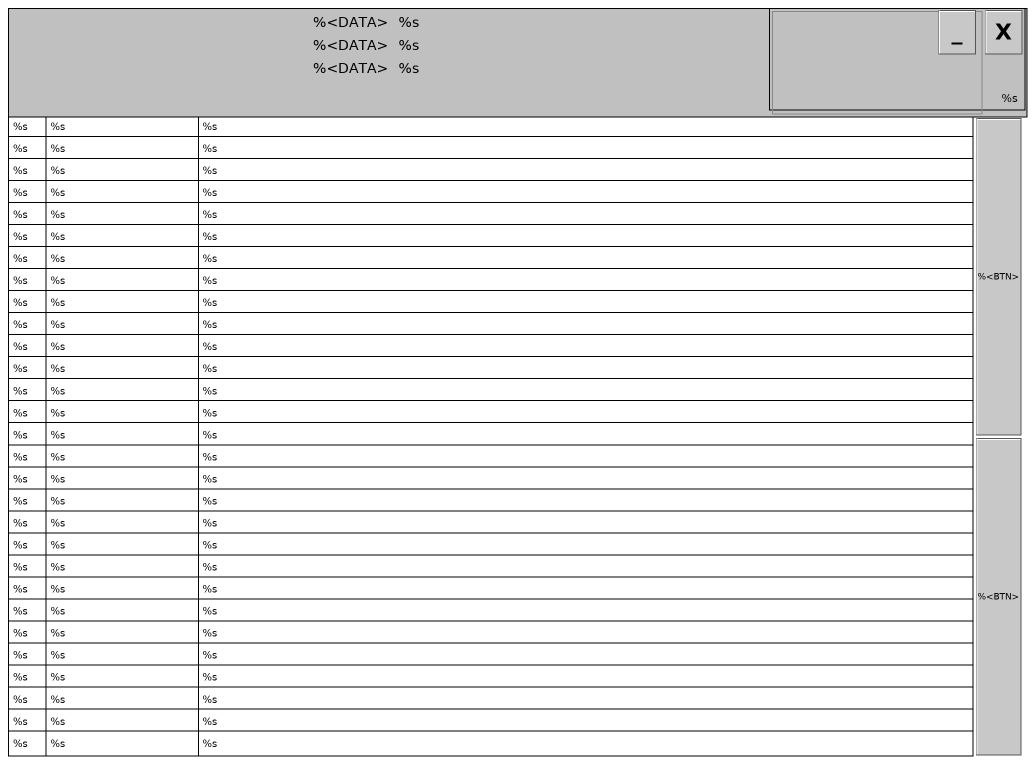
embedded screen at (4,112)-(969,754): zLib_ErrorList; opens ZOOMTOCALLER
button at (972,116)-(1017,433): text "%<BTN>"; shows 'up'; runs INTERN ASSIGN Visu.ErrorHistoryScroll:=(Visu.ErrorHistoryScroll - 29)
button at (972,436)-(1017,753): text "%<BTN>"; shows 'down'; runs INTERN ASSIGN Visu.ErrorHistoryScroll:=(Visu.ErrorHistoryScroll + 29)
rectangle at (0,114)-(971,765): opens ZOOMTOCALLER
rectangle at (248,50)-(387,67): shows 'TypeDescription'
rectangle at (889,87)-(1019,106): text "%s"; shows .gVarStrSystemTime
embedded screen at (933,8)-(1018,52): MIN_EXIT; invisible if TRUE
rectangle at (388,33)-(673,53): text "%s"; shows .TD.ArtNo
rectangle at (247,33)-(386,53): text "%<DATA>"; shows 'ArtNo'
rectangle at (388,10)-(673,30): text "%s"; shows .TD.TypeName
rectangle at (247,10)-(386,30): text "%<DATA>"; shows 'TypeName'
rectangle at (388,56)-(673,76): text "%s"; shows .TD.TypeDescription
rectangle at (247,56)-(386,76): text "%<DATA>"; shows 'TypeDescription'
3 more shapes without text or variables
*)

(* Visualisation SYSTEM_FEATURES
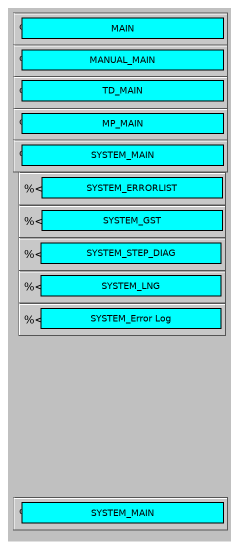
embedded screen at (3,115)-(226,648): M0003_System
*)

(* Visualisation SYSTEM_GST
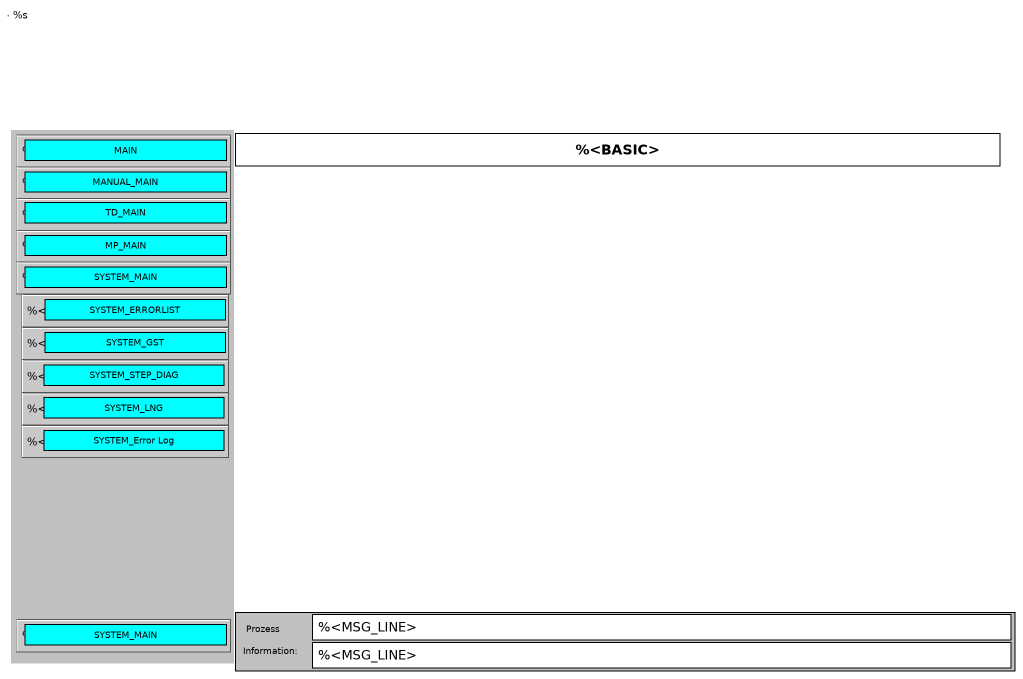
rectangle at (227,118)-(992,151): text "%<BASIC>"; shows 'Objekte ohne Grundstellung'
embedded screen at (3,115)-(226,648): M0003_System
rectangle at (227,597)-(1007,656): text "Prozess /  / Information:"
rectangle at (304,599)-(1003,625): text "%<MSG_LINE>"; shows ProcessMessage01
rectangle at (304,627)-(1003,653): text "%<MSG_LINE>"; shows ProcessMessage02
rectangle at (0,0)-(0,0): text "%s"; shows ListHomeNOK.HomeNOKArray[INDEX]
1 more shapes without text or variables
*)

(* Visualisation SYSTEM_LNG
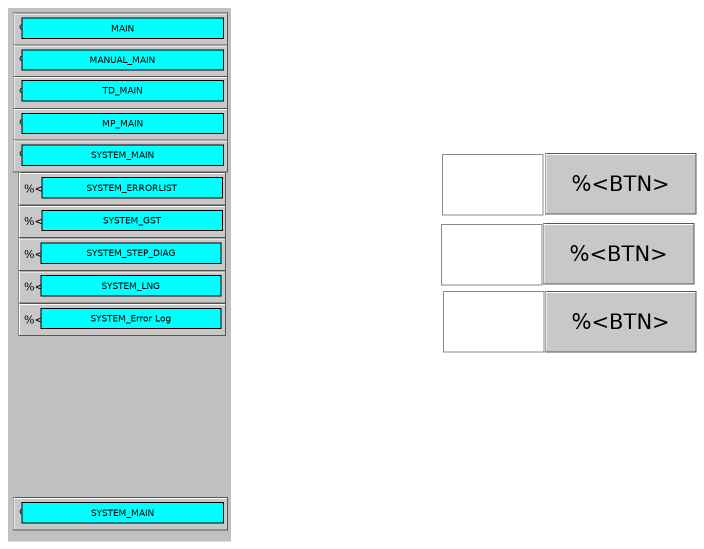
embedded screen at (3,115)-(226,648): M0003_System
other_BMP at (437,261)-(538,322): taps ST_Lng.btn_Language[0].tasten; runs INTERN LANGUAGE de
other_BMP at (436,331)-(537,392): taps ST_Lng.btn_Language[1].tasten; runs INTERN LANGUAGE en
other_BMP at (438,398)-(539,459): taps ST_Lng.btn_Language[2].tasten; runs INTERN LANGUAGE cz
button at (540,260)-(691,321): text "%<BTN>"; shows ST_Lng.btn_Language[0].Text; taps ST_Lng.btn_Language[0].tasten; runs INTERN LANGUAGE DE; dynamic style ST_Lng.btn_Language[0].innenFarbe
button at (538,330)-(689,391): text "%<BTN>"; shows ST_Lng.btn_Language[1].Text; taps ST_Lng.btn_Language[1].tasten; runs INTERN LANGUAGE EN; dynamic style ST_Lng.btn_Language[1].innenFarbe
button at (540,398)-(691,459): text "%<BTN>"; shows ST_Lng.btn_Language[2].Text; taps ST_Lng.btn_Language[2].tasten; runs INTERN LANGUAGE CZ; dynamic style ST_Lng.btn_Language[2].innenFarbe
*)

(* Visualisation SYSTEM_MAIN
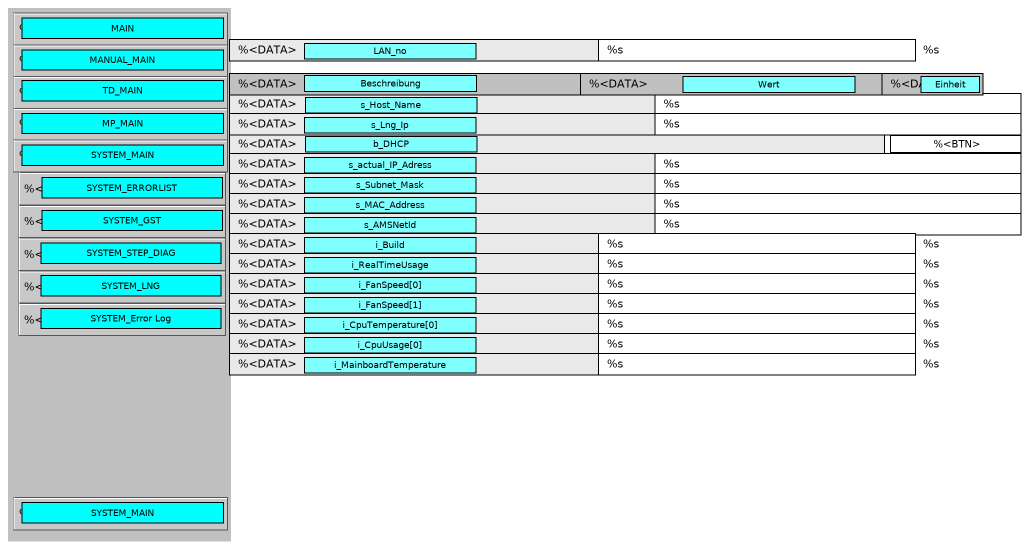
embedded screen at (3,115)-(226,648): M0003_System
embedded screen at (224,200)-(1016,222): Data_LINE_STR
embedded screen at (224,240)-(1016,262): DATA_LINE_B
rectangle at (300,204)-(472,220): text "s_Host_Name"; invisible if TRUE
rectangle at (300,243)-(472,259): text "b_DHCP"; invisible if TRUE
embedded screen at (224,260)-(1016,282): DATA_LINE_STR
rectangle at (299,264)-(471,280): text "s_actual_IP_Adress"; invisible if TRUE
embedded screen at (224,280)-(1016,302): DATA_LINE_STR
rectangle at (299,284)-(471,300): text "s_Subnet_Mask"; invisible if TRUE
embedded screen at (224,300)-(1016,322): DATA_LINE_STR
rectangle at (299,304)-(471,320): text "s_MAC_Address"; invisible if TRUE
embedded screen at (224,320)-(1016,342): DATA_LINE_STR
rectangle at (299,324)-(471,340): text "s_AMSNetId"; invisible if TRUE
embedded screen at (224,340)-(1016,362): Data_LINE_i16
rectangle at (299,344)-(471,360): text "i_Build"; invisible if TRUE
embedded screen at (224,360)-(1016,382): Data_LINE_i16
rectangle at (299,364)-(471,380): text "i_RealTimeUsage"; invisible if TRUE
embedded screen at (224,380)-(1016,402): Data_LINE_i16
rectangle at (299,384)-(471,400): text "i_FanSpeed[0]"; invisible if TRUE
embedded screen at (224,400)-(1016,422): Data_LINE_i16
rectangle at (299,404)-(471,420): text "i_FanSpeed[1]"; invisible if TRUE
embedded screen at (224,420)-(1016,442): Data_LINE_i16
rectangle at (299,424)-(471,440): text "i_CpuTemperature[0]"; invisible if TRUE
embedded screen at (224,440)-(1016,462): Data_LINE_i16
rectangle at (299,444)-(471,460): text "i_CpuUsage[0]"; invisible if TRUE
embedded screen at (224,460)-(1016,482): Data_LINE_i16
rectangle at (299,464)-(471,480): text "i_MainboardTemperature"; invisible if TRUE
embedded screen at (224,180)-(978,202): DATA_HEADER
embedded screen at (224,220)-(1016,242): DATA_LINE_STR
rectangle at (299,224)-(471,240): text "s_Lng_Ip"; invisible if TRUE
embedded screen at (224,146)-(1016,168): Data_LINE_i16
rectangle at (299,150)-(471,166): text "LAN_no"; invisible if TRUE
*)

(* Visualisation SYSTEM_STEP_DIAG
